// TwinCAT 3 PLC project ReadCSV
// ProgramVersion: 3.1.4022.4
// libraries:
//   Tc2_Standard, * (Beckhoff Automation GmbH)
//   Tc2_System, * (Beckhoff Automation GmbH)
//   Tc2_Utilities, * (Beckhoff Automation GmbH)
//   Tc3_Module, * (Beckhoff Automation GmbH)
// project tree:
//   DUTs/ eCSVFileReadStep.TcDUT, E_ReadCSVStep.TcDUT
//   GVLs/ GVL_General.TcGVL
//   / PlcTask.TcTTO
//   POUs/ FB_Blinking.TcPOU, MAIN.TcPOU, ReadCSV.TcPOU, ReadCSVSecondPractice.TcPOU
// real-time tasks:
//   TASK PlcTask: cycle T#10ms, priority 20, ADS port 350

CONFIGURATION ReadCSV
    RESOURCE PLC ON TwinCAT3
        TASK PlcTask(INTERVAL := T#10ms, PRIORITY := 20);
        PROGRAM MAIN WITH PlcTask : MAIN;
    END_RESOURCE
END_CONFIGURATION

// ---- DUTs/eCSVFileReadStep.TcDUT
{attribute 'qualified_only'}
{attribute 'strict'}
TYPE eCSVFileReadStep :
(
	iStep_Init := 0,
	iStep_Open,
	iStep_OpenWait,
	iStep_ReadSingleLine,
	iStep_ReadSingleWait,
	iStep_ParseSingleLine,	
	iStep_CloseOrError
	
);
END_TYPE

// ---- DUTs/E_ReadCSVStep.TcDUT
{attribute 'qualified_only'}
{attribute 'strict'}
TYPE E_ReadCSVStep :
(
	Step_Init := 0,
	Step_Open	:= 10,	
	Step_OpenWaite		:= 20,
	Step_ReadSingleLine		:= 30,
	Step_ReadSingleLineWait	,
	Step_ParseSingleLine,
	Step_Close	,
	Step_ErrorOrEnd		:= 999
);
END_TYPE

// ---- GVLs/GVL_General.TcGVL
{attribute 'qualified_only'}
VAR_GLOBAL
	
	database: ARRAY[0..MAX_CSV_ROWS, 0..MAX_CSV_COLUMNS] OF STRING;
	
	dataArray: ARRAY[0..MAX_CSV_ROWS, 0..MAX_CSV_COLUMNS] OF STRING;
END_VAR

VAR_GLOBAL CONSTANT
	MAX_CSV_COLUMNS			:INT:=99;
	MAX_CSV_ROWS			: INT:=99;
END_VAR

// ---- POUs/MAIN.TcPOU
PROGRAM MAIN
VAR
	bChangeSeparatorToComma: BOOL;
	fbBlink		:FB_Blinking;
	bBlink			:BOOL;
	bBlink2			:BOOL;
	
	ton2		:TON;
END_VAR

IF bChangeSeparatorToComma THEN
	DEFAULT_CSV_FIELD_SEP := 16#2C;(* Comma ASCII code *)
ELSE
	DEFAULT_CSV_FIELD_SEP := 16#3B;(* Semicolon ASCII code *)
END_IF



	//ReadCSV();
	
	//ReadCSVSecondPractice();

	//fbBlink.M_Blink();
	
	 
	
	//bBlink := NOT bBlink;
	
	
	
	
	ton2(IN:= NOT ton2.Q, PT:=T#0.5S , Q=> , ET=> );


	IF	ton2.Q THEN 
		ton2(IN:= FALSE);
		bBlink2 := NOT bBlink2;
	END_IF

END_PROGRAM

// ---- POUs/FB_Blinking.TcPOU
FUNCTION_BLOCK FB_Blinking
VAR_INPUT
END_VAR
VAR_OUTPUT	
	
END_VAR
VAR
	ton1		:TON;
END_VAR

METHOD M_Blink : BOOL
VAR_OUTPUT
	bBlink		:BOOL;
END_VAR
ton1(IN:= NOT ton1.Q, PT:= T#1S, Q=> , ET=> );

IF	ton1.Q THEN
	ton1(IN:= FALSE, PT:= T#1S, Q=> , ET=> );	
	bBlink := NOT bBlink;
END_IF
END_METHOD

END_FUNCTION_BLOCK

// ---- POUs/ReadCSV.TcPOU
PROGRAM ReadCSV
VAR
		
	sFileName		:STRING:='C:\Temp\TextModeGen.csv';
	
	fbFileOpen: FB_FileOpen;
	//fbFilePuts: FB_FilePuts;
	fbFileGets: FB_FileGets;
	fbFileClose: FB_FileClose;
	bRead			:BOOL;
	iStep			:E_ReadCSVStep;
	sCSVLine		:T_MaxString;
	fbReader: FB_CSVMemBufferReader;
	sCSVField		:T_MaxString;
	nRow			:INT:=0;
	nColumn			:INT:=0;
	hFile			:UINT;
	bBusy			:BOOL;
END_VAR

CASE iStep OF
	E_ReadCSVStep.Step_Init:	
		IF	bRead THEN 
			bRead := FALSE;	
			bBusy := TRUE;
			hFile := 0;
			nRow := 0;
			nColumn := 0;
			MEMSET(ADR(GVL_General.database),0, SIZEOF(GVL_General.database));			
			iStep:=	E_ReadCSVStep.Step_Open;			
		END_IF
		
	E_ReadCSVStep.Step_Open: (*open source file*)
		fbFileOpen(sNetId:= ,sPathName:= ,nMode:= ,ePath:= ,bExecute:=FALSE,
					tTimeout:=T#3S ,bBusy=> ,bError=> ,nErrId=> ,hFile=> );
					
		fbFileOpen(sNetId:= ,sPathName:= sFileName, nMode:= FOPEN_MODEREAD  ,ePath:=PATH_GENERIC ,bExecute:=TRUE,
					tTimeout:=T#3S ,bBusy=> ,bError=> ,nErrId=> ,hFile=>hFile);
		
		iStep := E_ReadCSVStep.Step_OpenWaite;
		
	E_ReadCSVStep.Step_OpenWaite:  (* confirm the open action*)
	
		fbFileOpen(sNetId:= ,sPathName:= sFileName, nMode:= FOPEN_MODEREAD  ,ePath:=PATH_GENERIC ,bExecute:=FALSE,
					tTimeout:=T#3S ,bBusy=> ,bError=> ,nErrId=> ,hFile=>hFile);
		IF NOT fbFileOpen.bBusy THEN 
			IF NOT fbFileOpen.bError THEN 
				iStep := E_ReadCSVStep.Step_ReadSingleLine;
			ELSE	(*error file not found?*)
				iStep := E_ReadCSVStep.Step_ErrorOrEnd;
			END_IF			
		END_IF
		
	E_ReadCSVStep.Step_ReadSingleLine:
		fbFileGets(sNetId:= ,hFile:= ,bExecute:=FALSE,tTimeout:=,bBusy=> ,bError=> ,nErrId=> ,sLine=> ,bEOF=> );
		
		fbFileGets(sNetId:= ,hFile:=hFile ,bExecute:=TRUE,tTimeout:=T#3S,
					bBusy=> ,bError=> ,nErrId=> ,sLine=>sCSVLine ,bEOF=> );
		
		iStep := E_ReadCSVStep.Step_ReadSingleLineWait;
		
	E_ReadCSVStep.Step_ReadSingleLineWait:(*wait until fbFileGets not busy*)
		fbFileGets(sNetId:= ,hFile:=hFile ,bExecute:=FALSE,tTimeout:=T#3S,
					bBusy=> ,bError=> ,nErrId=> ,sLine=>sCSVLine ,bEOF=> );
		
		IF NOT fbFileGets.bBusy THEN 
			IF NOT fbFileGets.bError THEN 
				IF fbFileGets.bEOF THEN
					iStep := E_ReadCSVStep.Step_Close; (* end of the file, then close the source file*)
				ELSE 
					(* FB_FileGets returns text line without the CR (carriage return) character.
					We have to restore the CR character (replace the $L character with $R$L characters) *)
					IF RIGHT(sCSVLine,1) = '$L' THEN 
						sCSVLine := REPLACE(STR1:= sCSVLine,STR2:= '$R$L', P:= LEN(STR:= sCSVLine),L:=2);
					END_IF
					iStep := E_ReadCSVStep.Step_ParseSingleLine;
				END_IF	
			ELSE
				iStep:= E_ReadCSVStep.Step_ErrorOrEnd;			
			END_IF
		END_IF  
		
	E_ReadCSVStep.Step_ParseSingleLine:
			
		fbReader.eCmd := eEnumCmd_First; (*Read first field value*)
		REPEAT
			fbReader(pBuffer:=ADR(sCSVLine) ,cbBuffer:= SIZEOF(sCSVLine),bOk=> ,getValue=>sCSVField ,pValue=> ,cbValue=> ,bCRLF=> ,cbRead=> );			
			IF fbReader.bOk THEN 
				fbReader.eCmd := eEnumCmd_Next;	
					IF(nRow <= GVL_General.MAX_CSV_ROWS) THEN 
						IF(nColumn <= GVL_General.MAX_CSV_COLUMNS) THEN 
							GVL_General.database[nRow,nColumn] := CSVFIELD_TO_STRING(in:= sCSVField,bQM:= FALSE);
						END_IF
					END_IF			
			
				nColumn := nColumn + 1;
				IF(fbReader.bCRLF) THEN 
					nColumn := 0;
					nRow := nRow + 1;					
				END_IF
			ELSE	
				iStep:= E_ReadCSVStep.Step_ReadSingleLine;
			END_IF		
		UNTIL NOT fbReader.bOk	
		END_REPEAT
		
	E_ReadCSVStep.Step_Close: (*close the source file*)
	
		fbFileClose(bExecute:= FALSE);		
		fbFileClose(sNetId:= ,hFile:=hFile ,bExecute:= TRUE,tTimeout:=T#3S ,bBusy=> ,bError=> ,nErrId=> );		
		IF NOT	fbFileClose.bBusy THEN 
			IF	NOT fbFileClose.bError THEN 
				hFile := 0;
				iStep := E_ReadCSVStep.Step_ErrorOrEnd;
			END_IF
		END_IF
		
	E_ReadCSVStep.Step_ErrorOrEnd:
		IF (hFile <> 0) THEN 
			iStep := E_ReadCSVStep.Step_Close;
		ELSE
			bBusy := FALSE;
			iStep := E_ReadCSVStep.Step_Init;
		END_IF	
		
END_CASE

END_PROGRAM

// ---- POUs/ReadCSVSecondPractice.TcPOU
PROGRAM ReadCSVSecondPractice
VAR
	
	iStep		:eCSVFileReadStep;
	nRow			:INT:=0;
	nColumn			:INT:=0;
	bRead			:BOOL;
	handleFile		:UINT;
	fbFileClose: FB_FileClose;
	fbFileGets: FB_FileGets;
	fbFileOpen: FB_FileOpen;
	fbRead: FB_CSVMemBufferReader;
	FilePath		:STRING:= 'C:\Temp\TextModeGen.csv';
	sCSVLine			:T_MaxString;
	bReadError: BOOL;
	sCSVField: T_MaxString;
END_VAR

CASE iStep OF
	eCSVFileReadStep.iStep_Init:
		IF	bRead THEN 
			bRead := FALSE;
			nRow := 0;
			nColumn := 0;
			MEMSET(ADR(GVL_General.dataArray),0,SIZEOF(GVL_General.dataArray));
			iStep := eCSVFileReadStep.iStep_Open;
		END_IF
		
	eCSVFileReadStep.iStep_Open:	(*prepare to open source file*)
		fbFileOpen(bExecute:=FALSE);
					
		fbFileOpen(sNetId:= ,sPathName:=FilePath ,nMode:= FOPEN_MODEREAD OR FOPEN_MODETEXT,ePath:=PATH_GENERIC ,bExecute:=TRUE,
					tTimeout:=T#3S ,bBusy=> ,bError=> ,nErrId=> ,hFile=> handleFile);
					
		iStep := eCSVFileReadStep.iStep_OpenWait;
		
	eCSVFileReadStep.iStep_OpenWait:

			fbFileOpen(sNetId:= ,sPathName:=FilePath ,nMode:= FOPEN_MODEREAD,ePath:=PATH_GENERIC ,bExecute:=FALSE,
					tTimeout:=T#3S ,bBusy=> ,bError=> ,nErrId=> ,hFile=> handleFile);	
		IF NOT fbFileOpen.bBusy THEN 
			IF NOT fbFileOpen.bError THEN 
				iStep := eCSVFileReadStep.iStep_ReadSingleLine;	
			ELSE
				iStep := eCSVFileReadStep.iStep_CloseOrError;
			END_IF
		END_IF
		
		
	eCSVFileReadStep.iStep_ReadSingleLine:
	
		fbFileGets(sNetId:= ,hFile:=handleFile,bExecute:=FALSE,tTimeout:=T#3S,
					bBusy=> ,bError=> ,nErrId=> ,sLine=> sCSVLine,bEOF=> );
					
		fbFileGets(sNetId:= ,hFile:=handleFile,bExecute:=TRUE,tTimeout:=T#3S,
					bBusy=> ,bError=> ,nErrId=> ,sLine=>sCSVLine,bEOF=> );
					
		iStep := eCSVFileReadStep.iStep_ReadSingleWait;


	(*eCSVFileReadStep.iStep_ReadSingleWait:		
		fbFileGets(sNetId:= ,hFile:=handleFile,bExecute:=FALSE,tTimeout:=T#3S,
					bBusy=> ,bError=> ,nErrId=> ,sLine=> sCSVLine,bEOF=> );	
					
		IF NOT fbFileGets.bBusy THEN 
			IF NOT fbFileGets.bError THEN 
				IF fbFileGets.bEOF THEN 
					iStep := eCSVFileReadStep.iStep_CloseOrError;
				END_IF
				//add CRLF to the end of the CSVField
				IF(RIGHT(sCSVLine,1) = '$N') THEN 
					sCSVLine := REPLACE(sCSVLine,'$R$N',2,Len(sCSVLine));
					iStep := eCSVFileReadStep.iStep_ParseSingleLine;
				END_IF				
			ELSE
				iStep := eCSVFileReadStep.iStep_CloseOrError;
			END_IF
		END_IF*)
		
		
	eCSVFileReadStep.iStep_ReadSingleWait:		
		fbFileGets(sNetId:= ,hFile:=handleFile,bExecute:=FALSE,tTimeout:=T#3S,
					bBusy=> ,bError=> ,nErrId=> ,sLine=> sCSVLine,bEOF=> );	
					
		IF NOT fbFileGets.bBusy THEN 
			IF NOT fbFileGets.bError THEN 
				IF fbFileGets.bEOF THEN 
					iStep := eCSVFileReadStep.iStep_CloseOrError;
				ELSE
				//add CRLF to the end of the CSVField
					IF(RIGHT(sCSVLine,1) = '$N') THEN 
						sCSVLine := REPLACE(sCSVLine,'$R$N',2,Len(sCSVLine));
						iStep := eCSVFileReadStep.iStep_ParseSingleLine;
					END_IF	
				END_IF			
			ELSE
				iStep := eCSVFileReadStep.iStep_CloseOrError;
			END_IF
		END_IF
		
	eCSVFileReadStep.iStep_ParseSingleLine:
		fbRead.eCmd := eEnumCmd_First;
		REPEAT
			fbRead(pBuffer:=ADR(sCSVLine),cbBuffer:=SIZEOF(sCSVLine),bOk=> , 
					getValue=>sCSVField ,pValue=> ,cbValue=>,bCRLF=> ,cbRead=> );			
			IF	fbRead.bOk THEN 
				fbRead.eCmd := eEnumCmd_Next;
				IF(nRow < GVL_General.MAX_CSV_ROWS) THEN
					IF (nColumn < GVL_General.MAX_CSV_COLUMNS) THEN 
						GVL_General.dataArray[nRow,nColumn] := CSVFIELD_TO_STRING(in:= sCSVField, bQM:= FALSE);											
					END_IF					
				END_IF
				nColumn := nColumn +1;	
				IF(fbRead.bCRLF) THEN 
					nColumn := 0;
					nRow 	:= nRow + 1;
				END_IF
			ELSE
				iStep := eCSVFileReadStep.iStep_ReadSingleLine;
			END_IF			
		UNTIL NOT fbRead.bOk
		END_REPEAT		
		
		
	eCSVFileReadStep.iStep_CloseOrError:
		fbFileClose(sNetId:= ,hFile:=handleFile ,bExecute:=FALSE,tTimeout:= ,bBusy=> ,bError=> ,nErrId=> );
		fbFileClose(sNetId:= ,hFile:=handleFile ,bExecute:=TRUE,tTimeout:= ,bBusy=> ,bError=> ,nErrId=> );
		IF NOT fbFileClose.bBusy THEN 
			IF NOT fbFileClose.bError THEN 

				iStep := eCSVFileReadStep.iStep_Init;
			ELSE
				bReadError := TRUE;
			END_IF
		END_IF	
END_CASE

END_PROGRAM
